ABB RAPID module: RapidProgrammeCode.mod

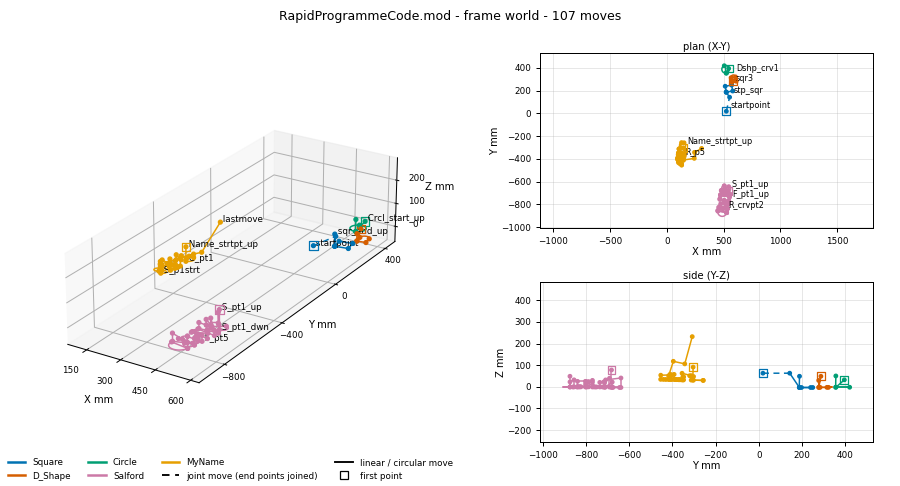
[picture p0: tool path of RapidProgrammeCode.mod in frame world, 107 of 113 moves have a stored position in this frame; points joined in program order, loops and branches not executed]
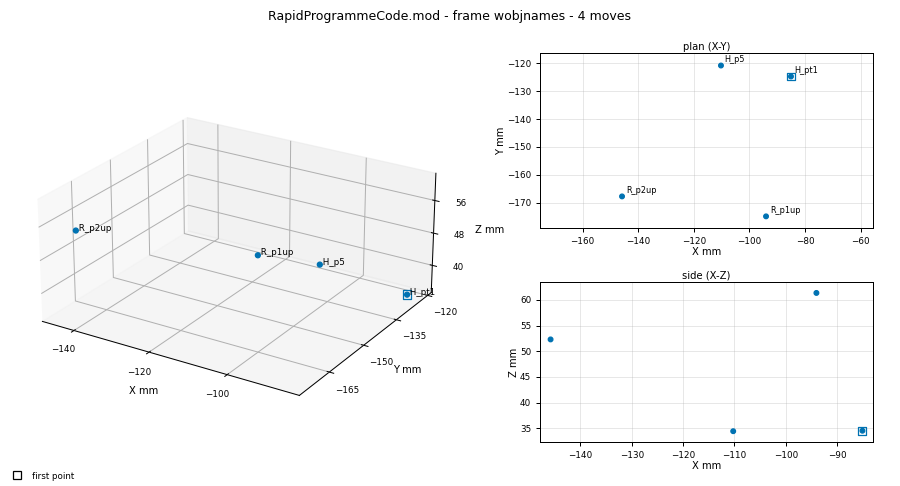
[picture p1: tool path of RapidProgrammeCode.mod in frame wobjnames, 4 of 113 moves have a stored position in this frame; points joined in program order, loops and branches not executed]
MODULE Module1
TASK PERS tooldata toolpen:=[TRUE,[[100,0,20],[1,0,0,0]],[0.1,[50,0,10],[1,0,0,0],0,0,0]];
TASK PERS wobjdata wobjshapes:=[FALSE,TRUE,"",[[456.883,136.274,-5.92371],[0.996185,0.000008375,-0.000001296,0.0872714]],[[0,0,0],[1,0,0,0]]];
CONST robtarget pointoforigin:=[[581.51,18.36,14.08],[0.66738,-0.167376,0.708898,0.155091],[-1,-1,0,1],[9E+9,9E+9,9E+9,9E+9,9E+9,9E+9]];
TASK PERS wobjdata wobjsalf:=[FALSE,TRUE,"",[[460.965,-385.411,-5.78367],[1,-0.000000822,-0.000000764,-0.000000546]],[[0,0,0],[1,0,0,0]]];
TASK PERS wobjdata wobjname:=[FALSE,TRUE,"",[[241.141,-193.884,-5.92118],[0.999813,-0.0119256,-0.000182929,0.0152539]],[[0,0,0],[1,0,0,0]]];
CONST robtarget startpoint:=[[45.66,-127.08,69.03],[0.678366,-0.104877,0.720803,0.0962504],[-1,-1,0,1],[9E+09,9E+09,9E+09,9E+09,9E+09,9E+09]];
CONST robtarget startpoint10:=[[105.53,42.34,81.65],[0.678367,-0.104876,0.720802,0.0962504],[0,-1,0,1],[9E+9,9E+9,9E+9,9E+9,9E+9,9E+9]];
CONST robtarget stp_sqr:=[[95.33,-10.14,69.03],[0.678365,-0.104877,0.720803,0.0962505],[0,-1,0,1],[9E+09,9E+09,9E+09,9E+09,9E+09,9E+09]];
CONST robtarget stp_sqr10:=[[72.90,39.01,0.49],[0.678366,-0.104876,0.720802,0.0962504],[0,-1,-1,1],[9E+9,9E+9,9E+9,9E+9,9E+9,9E+9]];
CONST robtarget stp_sqr1:=[[72.90,39.01,0.49],[0.678366,-0.104876,0.720802,0.0962504],[0,-1,-1,1],[9E+9,9E+9,9E+9,9E+9,9E+9,9E+9]];
CONST robtarget stp_sqr11:=[[131.10,38.55,0.49],[0.678367,-0.104876,0.720802,0.0962505],[0,-1,0,1],[9E+9,9E+9,9E+9,9E+9,9E+9,9E+9]];
CONST robtarget stp_sqr2:=[[131.10,38.55,0.49],[0.678367,-0.104876,0.720802,0.0962505],[0,-1,0,1],[9E+9,9E+9,9E+9,9E+9,9E+9,9E+9]];
CONST robtarget stp_sqr12:=[[130.95,91.71,0.49],[0.678366,-0.104876,0.720802,0.0962506],[0,-1,0,1],[9E+9,9E+9,9E+9,9E+9,9E+9,9E+9]];
CONST robtarget stp_sqr3:=[[130.95,91.71,0.49],[0.678366,-0.104876,0.720802,0.0962506],[0,-1,0,1],[9E+9,9E+9,9E+9,9E+9,9E+9,9E+9]];
CONST robtarget stp_sqr13:=[[72.83,91.46,0.49],[0.678365,-0.104877,0.720803,0.0962506],[0,-1,-1,1],[9E+9,9E+9,9E+9,9E+9,9E+9,9E+9]];
CONST robtarget stp_sqr4:=[[72.83,91.46,0.49],[0.678365,-0.104877,0.720803,0.0962506],[0,-1,-1,1],[9E+9,9E+9,9E+9,9E+9,9E+9,9E+9]];
CONST robtarget sqr1:=[[73.63,39.09,2.89],[0.678366,-0.104876,0.720803,0.0962505],[0,-1,-1,1],[9E+09,9E+09,9E+09,9E+09,9E+09,9E+09]];
CONST robtarget sqr2:=[[131.71,38.69,2.89],[0.678366,-0.104876,0.720803,0.0962504],[0,-1,0,1],[9E+09,9E+09,9E+09,9E+09,9E+09,9E+09]];
CONST robtarget sqr3:=[[131.6,91.52,2.89],[0.678365,-0.104877,0.720803,0.0962505],[0,-1,0,1],[9E+09,9E+09,9E+09,9E+09,9E+09,9E+09]];
CONST robtarget sqr4:=[[74.02,91.72,2.89],[0.678364,-0.104877,0.720805,0.0962503],[0,-1,-1,1],[9E+09,9E+09,9E+09,9E+09,9E+09,9E+09]];
CONST robtarget sqr14:=[[75.15,37.61,0.49],[0.678366,-0.104877,0.720803,0.0962507],[0,-1,-1,1],[9E+9,9E+9,9E+9,9E+9,9E+9,9E+9]];
CONST robtarget sqr24:=[[75.29,39.68,0.49],[0.678366,-0.104877,0.720803,0.0962508],[0,-1,-1,1],[9E+9,9E+9,9E+9,9E+9,9E+9,9E+9]];
CONST robtarget sqr5:=[[75.37,38.14,2.89],[0.678365,-0.104877,0.720804,0.0962503],[0,-1,-1,1],[9E+09,9E+09,9E+09,9E+09,9E+09,9E+09]];
CONST robtarget sqr15:=[[73.98,39.56,54.84],[0.678365,-0.104877,0.720803,0.0962503],[0,-1,0,1],[9E+9,9E+9,9E+9,9E+9,9E+9,9E+9]];
CONST robtarget sqr25:=[[73.98,39.56,54.84],[0.678365,-0.104877,0.720803,0.0962503],[0,-1,0,1],[9E+9,9E+9,9E+9,9E+9,9E+9,9E+9]];
CONST robtarget sqr_end_up:=[[73.98,39.56,54.84],[0.678365,-0.104877,0.720803,0.0962503],[0,-1,0,1],[9E+09,9E+09,9E+09,9E+09,9E+09,9E+09]];
CONST robtarget sqr_end_up10:=[[152.51,126.22,54.84],[0.678365,-0.104877,0.720804,0.0962505],[0,-1,-1,1],[9E+9,9E+9,9E+9,9E+9,9E+9,9E+9]];
CONST robtarget Dshp_start_up:=[[152.51,126.22,54.84],[0.678365,-0.104877,0.720804,0.0962505],[0,-1,-1,1],[9E+09,9E+09,9E+09,9E+09,9E+09,9E+09]];
CONST robtarget Dshp_start_up10:=[[139.65,118.70,3.57],[0.678364,-0.104877,0.720804,0.0962503],[0,-1,-1,1],[9E+9,9E+9,9E+9,9E+9,9E+9,9E+9]];
CONST robtarget Dshp_pt1:=[[139.65,118.7,3.57],[0.678364,-0.104877,0.720804,0.0962503],[0,-1,-1,1],[9E+09,9E+09,9E+09,9E+09,9E+09,9E+09]];
CONST robtarget Dshp_pt11:=[[177.47,117.91,3.57],[0.678365,-0.104877,0.720804,0.0962505],[0,-1,0,1],[9E+9,9E+9,9E+9,9E+9,9E+9,9E+9]];
CONST robtarget Dshp_pt2:=[[177.47,117.91,3.57],[0.678365,-0.104877,0.720804,0.0962505],[0,-1,0,1],[9E+09,9E+09,9E+09,9E+09,9E+09,9E+09]];
CONST robtarget Dshp_pt12:=[[177.53,157.32,3.57],[0.678364,-0.104877,0.720805,0.0962505],[0,0,-1,1],[9E+9,9E+9,9E+9,9E+9,9E+9,9E+9]];
CONST robtarget Dshp_pt3:=[[177.53,157.32,3.57],[0.678364,-0.104877,0.720805,0.0962505],[0,0,-1,1],[9E+09,9E+09,9E+09,9E+09,9E+09,9E+09]];
CONST robtarget Dshp_pt23:=[[138.50,156.89,3.57],[0.678363,-0.104877,0.720805,0.0962503],[0,0,-1,1],[9E+9,9E+9,9E+9,9E+9,9E+9,9E+9]];
CONST robtarget Dshp_pt13:=[[156.88,176.76,3.57],[0.678363,-0.104877,0.720805,0.0962503],[0,0,-1,1],[9E+9,9E+9,9E+9,9E+9,9E+9,9E+9]];
CONST robtarget Dshp_crv1:=[[156.88,176.76,3.57],[0.678363,-0.104877,0.720805,0.0962503],[0,0,-1,1],[9E+09,9E+09,9E+09,9E+09,9E+09,9E+09]];
CONST robtarget Dshp_crv2:=[[138.5,156.89,3.57],[0.678363,-0.104877,0.720805,0.0962503],[0,0,-1,1],[9E+09,9E+09,9E+09,9E+09,9E+09,9E+09]];
CONST robtarget Dshp_crv11:=[[139.05,118.30,3.57],[0.678363,-0.104877,0.720805,0.0962504],[0,-1,-1,1],[9E+9,9E+9,9E+9,9E+9,9E+9,9E+9]];
CONST robtarget Dshp_pt4:=[[139.05,118.3,3.57],[0.678363,-0.104877,0.720805,0.0962504],[0,-1,-1,1],[9E+09,9E+09,9E+09,9E+09,9E+09,9E+09]];
CONST robtarget Dshp_pt14:=[[139.05,118.30,35.44],[0.678363,-0.104877,0.720805,0.0962504],[0,-1,-1,1],[9E+9,9E+9,9E+9,9E+9,9E+9,9E+9]];
CONST robtarget Dshp_end_up:=[[139.05,118.3,35.44],[0.678363,-0.104877,0.720805,0.0962504],[0,-1,-1,1],[9E+09,9E+09,9E+09,9E+09,9E+09,9E+09]];
CONST robtarget Dshp_end_up10:=[[131.01,240.02,38.32],[0.678365,-0.104877,0.720803,0.0962513],[0,0,-1,1],[9E+9,9E+9,9E+9,9E+9,9E+9,9E+9]];
CONST robtarget Crcl_start_up:=[[131.01,240.02,38.32],[0.678365,-0.104877,0.720803,0.0962513],[0,0,-1,1],[9E+09,9E+09,9E+09,9E+09,9E+09,9E+09]];
CONST robtarget Crcl_start_up10:=[[104.28,205.24,4.07],[0.678363,-0.104878,0.720805,0.096251],[0,0,-1,1],[9E+9,9E+9,9E+9,9E+9,9E+9,9E+9]];
CONST robtarget Crcl_start_pt1:=[[104.28,205.24,4.07],[0.678363,-0.104878,0.720805,0.096251],[0,0,-1,1],[9E+09,9E+09,9E+09,9E+09,9E+09,9E+09]];
CONST robtarget Crcl_start_pt21:=[[97.32,270.88,4.07],[0.678363,-0.104878,0.720805,0.096251],[0,0,-1,1],[9E+9,9E+9,9E+9,9E+9,9E+9,9E+9]];
CONST robtarget Crcl_start_pt11:=[[134.47,246.88,4.07],[0.678363,-0.104878,0.720805,0.0962509],[0,0,-1,1],[9E+9,9E+9,9E+9,9E+9,9E+9,9E+9]];
CONST robtarget Crcl_pt2:=[[134.47,246.88,4.07],[0.678363,-0.104878,0.720805,0.0962509],[0,0,-1,1],[9E+09,9E+09,9E+09,9E+09,9E+09,9E+09]];
CONST robtarget Crcl_pt3:=[[97.32,270.88,4.07],[0.678363,-0.104878,0.720805,0.096251],[0,0,-1,1],[9E+09,9E+09,9E+09,9E+09,9E+09,9E+09]];
CONST robtarget Crcl_pt22:=[[104.26,203.85,4.07],[0.678363,-0.104878,0.720805,0.0962515],[0,0,-1,1],[9E+9,9E+9,9E+9,9E+9,9E+9,9E+9]];
CONST robtarget Crcl_pt12:=[[71.11,230.12,4.07],[0.678363,-0.104878,0.720805,0.0962513],[0,0,-1,1],[9E+9,9E+9,9E+9,9E+9,9E+9,9E+9]];
CONST robtarget Crcl_pt4:=[[71.11,230.12,4.07],[0.678363,-0.104878,0.720805,0.0962513],[0,0,-1,1],[9E+09,9E+09,9E+09,9E+09,9E+09,9E+09]];
CONST robtarget Crcl_pt5:=[[104.26,203.85,4.07],[0.678363,-0.104878,0.720805,0.0962515],[0,0,-1,1],[9E+09,9E+09,9E+09,9E+09,9E+09,9E+09]];
CONST robtarget Crcl_pt14:=[[103.87,204.92,56.32],[0.678365,-0.104876,0.720803,0.0962504],[0,0,-1,1],[9E+9,9E+9,9E+9,9E+9,9E+9,9E+9]];
CONST robtarget Crcl_end_up:=[[103.87,204.92,56.32],[0.678365,-0.104876,0.720803,0.0962504],[0,0,-1,1],[9E+09,9E+09,9E+09,9E+09,9E+09,9E+09]];
VAR num MyChoice:=0;
CONST robtarget Crcl_end_up10:=[[77.92,-295.75,83.77],[0.678363,-0.104878,0.720805,0.0962498],[-1,-1,0,1],[9E+9,9E+9,9E+9,9E+9,9E+9,9E+9]];
CONST robtarget S_pt1_up:=[[77.92,-295.75,83.77],[0.678363,-0.104878,0.720805,0.0962498],[-1,-1,0,1],[9E+09,9E+09,9E+09,9E+09,9E+09,9E+09]];
CONST robtarget S_pt1_up10:=[[77.92,-295.75,5.22],[0.678363,-0.104878,0.720805,0.0962496],[-1,-1,0,1],[9E+9,9E+9,9E+9,9E+9,9E+9,9E+9]];
CONST robtarget S_pt1_dwn:=[[77.92,-295.75,2.89],[0.678363,-0.104878,0.720805,0.0962498],[-1,-1,0,1],[9E+09,9E+09,9E+09,9E+09,9E+09,9E+09]];
CONST robtarget S_pt1_dwn20:=[[84.34,-258.56,5.22],[0.678363,-0.104877,0.720806,0.0962498],[-1,-1,0,1],[9E+9,9E+9,9E+9,9E+9,9E+9,9E+9]];
CONST robtarget S_pt1_dwn10:=[[100.17,-280.53,5.22],[0.678363,-0.104878,0.720805,0.0962498],[-1,-1,0,1],[9E+9,9E+9,9E+9,9E+9,9E+9,9E+9]];
CONST robtarget S_pt2_crv:=[[100.97,-278.71,2.9],[0.678364,-0.104879,0.720804,0.0962497],[-1,-1,0,1],[9E+09,9E+09,9E+09,9E+09,9E+09,9E+09]];
CONST robtarget S_pt2_crv2:=[[84.34,-258.56,5.22],[0.678363,-0.104877,0.720806,0.0962498],[-1,-1,0,1],[9E+9,9E+9,9E+9,9E+9,9E+9,9E+9]];
CONST robtarget S_pt2_crv10:=[[38.36,-288.97,5.22],[0.678362,-0.104877,0.720806,0.0962497],[-1,-1,0,1],[9E+9,9E+9,9E+9,9E+9,9E+9,9E+9]];
CONST robtarget S_pt3_crv2:=[[84.01,-258.59,2.9],[0.678364,-0.104878,0.720804,0.0962498],[-1,-1,0,1],[9E+09,9E+09,9E+09,9E+09,9E+09,9E+09]];
CONST robtarget S_pt4:=[[40.74,-288.86,2.9],[0.678364,-0.104878,0.720804,0.0962498],[-1,-1,0,1],[9E+09,9E+09,9E+09,9E+09,9E+09,9E+09]];
CONST robtarget S_pt24:=[[44.83,-251.34,5.22],[0.678362,-0.104877,0.720806,0.0962497],[-1,-1,0,1],[9E+9,9E+9,9E+9,9E+9,9E+9,9E+9]];
CONST robtarget S_pt14:=[[22.78,-267.45,5.22],[0.678362,-0.104877,0.720806,0.0962498],[-1,-1,0,1],[9E+9,9E+9,9E+9,9E+9,9E+9,9E+9]];
CONST robtarget S_pt5_crv3:=[[22.75,-267.87,2.89],[0.678363,-0.104878,0.720805,0.0962498],[-1,-1,0,1],[9E+09,9E+09,9E+09,9E+09,9E+09,9E+09]];
CONST robtarget S_pt6_crv4:=[[44.86,-252.05,2.89],[0.678363,-0.104878,0.720805,0.09625],[-1,-1,0,1],[9E+09,9E+09,9E+09,9E+09,9E+09,9E+09]];
CONST robtarget S_pt5_crv13:=[[44.83,-251.34,37.85],[0.678362,-0.104877,0.720806,0.0962496],[-1,-1,0,1],[9E+9,9E+9,9E+9,9E+9,9E+9,9E+9]];
CONST robtarget S_end_up:=[[44.86,-252.05,46.77],[0.678363,-0.104878,0.720805,0.09625],[-1,-1,0,1],[9E+09,9E+09,9E+09,9E+09,9E+09,9E+09]];
CONST robtarget S_end_up10:=[[92.49,-322.94,37.85],[0.678363,-0.104877,0.720806,0.0962493],[-1,-1,0,1],[9E+9,9E+9,9E+9,9E+9,9E+9,9E+9]];
CONST robtarget S_end_up20:=[[92.49,-322.94,37.85],[0.678363,-0.104877,0.720806,0.0962493],[-1,-1,0,1],[9E+9,9E+9,9E+9,9E+9,9E+9,9E+9]];
CONST robtarget A_start_up:=[[92.49,-322.94,37.85],[0.678363,-0.104877,0.720806,0.0962493],[-1,-1,0,1],[9E+09,9E+09,9E+09,9E+09,9E+09,9E+09]];
CONST robtarget A_start_up10:=[[91.38,-324.75,5.35],[0.678363,-0.104877,0.720806,0.0962492],[-1,-1,0,1],[9E+9,9E+9,9E+9,9E+9,9E+9,9E+9]];
CONST robtarget A_start_pt1:=[[91.38,-324.75,5.35],[0.678363,-0.104877,0.720806,0.0962492],[-1,-1,0,1],[9E+09,9E+09,9E+09,9E+09,9E+09,9E+09]];
CONST robtarget A_start_pt11:=[[18.61,-292.43,5.35],[0.678364,-0.104878,0.720805,0.0962491],[-1,-1,0,1],[9E+9,9E+9,9E+9,9E+9,9E+9,9E+9]];
CONST robtarget A_pt2:=[[18.61,-292.43,5.35],[0.678364,-0.104878,0.720805,0.0962491],[-1,-1,0,1],[9E+09,9E+09,9E+09,9E+09,9E+09,9E+09]];
CONST robtarget A_pt12:=[[18.61,-292.43,27.82],[0.678364,-0.104877,0.720805,0.096249],[-1,-1,0,1],[9E+9,9E+9,9E+9,9E+9,9E+9,9E+9]];
CONST robtarget A_line1_up:=[[18.61,-292.43,27.82],[0.678364,-0.104877,0.720805,0.096249],[-1,-1,0,1],[9E+09,9E+09,9E+09,9E+09,9E+09,9E+09]];
CONST robtarget A_line1_up10:=[[91.72,-324.34,4.75],[0.678363,-0.104878,0.720806,0.0962488],[-1,-1,0,1],[9E+9,9E+9,9E+9,9E+9,9E+9,9E+9]];
CONST robtarget A_line2_strt:=[[91.72,-324.34,4.75],[0.678363,-0.104878,0.720806,0.0962488],[-1,-1,0,1],[9E+09,9E+09,9E+09,9E+09,9E+09,9E+09]];
CONST robtarget A_line2_strt10:=[[11.68,-330.33,4.75],[0.678362,-0.104877,0.720806,0.096249],[-1,-1,0,1],[9E+9,9E+9,9E+9,9E+9,9E+9,9E+9]];
CONST robtarget A_line2_stp:=[[11.68,-330.33,4.75],[0.678362,-0.104877,0.720806,0.096249],[-1,-1,0,1],[9E+09,9E+09,9E+09,9E+09,9E+09,9E+09]];
CONST robtarget A_line2_stp10:=[[11.68,-330.33,29.04],[0.678362,-0.104877,0.720806,0.0962488],[-1,-1,0,1],[9E+9,9E+9,9E+9,9E+9,9E+9,9E+9]];
CONST robtarget A_line2_endup:=[[11.68,-330.33,29.04],[0.678362,-0.104877,0.720806,0.0962488],[-1,-1,0,1],[9E+09,9E+09,9E+09,9E+09,9E+09,9E+09]];
CONST robtarget A_line2_endup10:=[[43.93,-327.74,25.23],[0.678361,-0.104877,0.720807,0.0962489],[-1,-1,0,1],[9E+9,9E+9,9E+9,9E+9,9E+9,9E+9]];
CONST robtarget A_crssline_up:=[[43.93,-327.74,25.23],[0.678361,-0.104877,0.720807,0.0962489],[-1,-1,0,1],[9E+09,9E+09,9E+09,9E+09,9E+09,9E+09]];
CONST robtarget A_crssline_up10:=[[43.93,-327.74,4.82],[0.678361,-0.104878,0.720807,0.0962489],[-1,-1,0,1],[9E+9,9E+9,9E+9,9E+9,9E+9,9E+9]];
CONST robtarget A_crssline_pt1:=[[43.93,-327.74,4.82],[0.678361,-0.104878,0.720807,0.0962489],[-1,-1,0,1],[9E+09,9E+09,9E+09,9E+09,9E+09,9E+09]];
CONST robtarget A_crssline_pt11:=[[46.49,-305.03,4.82],[0.678361,-0.104878,0.720808,0.0962489],[-1,-1,0,1],[9E+9,9E+9,9E+9,9E+9,9E+9,9E+9]];
CONST robtarget A_crssline_pt2:=[[46.49,-305.03,4.82],[0.67836,-0.104878,0.720808,0.096249],[-1,-1,0,1],[9E+09,9E+09,9E+09,9E+09,9E+09,9E+09]];
CONST robtarget A_crssline_pt12:=[[46.49,-305.03,45.39],[0.67836,-0.104878,0.720808,0.0962488],[-1,-1,0,1],[9E+9,9E+9,9E+9,9E+9,9E+9,9E+9]];
CONST robtarget A_end_up:=[[46.49,-305.03,45.39],[0.67836,-0.104878,0.720808,0.0962488],[-1,-1,0,1],[9E+09,9E+09,9E+09,9E+09,9E+09,9E+09]];
CONST robtarget A_end_up10:=[[91.77,-349.30,45.39],[0.678361,-0.104878,0.720808,0.0962487],[-1,-1,0,1],[9E+9,9E+9,9E+9,9E+9,9E+9,9E+9]];
CONST robtarget L_start_up:=[[90.88,-349.88,26.27],[0.67836,-0.104879,0.720808,0.0962479],[-1,-1,0,1],[9E+09,9E+09,9E+09,9E+09,9E+09,9E+09]];
CONST robtarget L_start_up10:=[[89.10,-349.57,5.90],[0.67836,-0.104878,0.720808,0.0962488],[-1,-1,0,1],[9E+9,9E+9,9E+9,9E+9,9E+9,9E+9]];
CONST robtarget L_start_pt1:=[[90.88,-349.88,5.25],[0.67836,-0.104879,0.720809,0.0962479],[-1,-1,0,1],[9E+09,9E+09,9E+09,9E+09,9E+09,9E+09]];
CONST robtarget L_start_pt11:=[[11.36,-337.10,5.90],[0.67836,-0.104878,0.720808,0.0962488],[-1,-1,0,1],[9E+9,9E+9,9E+9,9E+9,9E+9,9E+9]];
CONST robtarget L_pt2:=[[11.36,-337.10,5.90],[0.67836,-0.104878,0.720808,0.0962488],[-1,-1,0,1],[9E+9,9E+9,9E+9,9E+9,9E+9,9E+9]];
CONST robtarget L_pt3_dwn:=[[11.26,-336.76,5.25],[0.67836,-0.104879,0.720809,0.0962477],[-1,-1,0,1],[9E+09,9E+09,9E+09,9E+09,9E+09,9E+09]];
CONST robtarget L_pt3_dwn10:=[[6.45,-364.89,29.17],[0.678361,-0.104878,0.720808,0.0962485],[-1,-1,0,1],[9E+9,9E+9,9E+9,9E+9,9E+9,9E+9]];
CONST robtarget L_pt3_up:=[[6.26,-365.07,5.25],[0.67836,-0.104879,0.720808,0.0962476],[-1,-1,0,1],[9E+9,9E+9,9E+9,9E+9,9E+9,9E+9]];
CONST robtarget L_pt3_up10:=[[82.67,-383.82,35.68],[0.678359,-0.104878,0.720809,0.0962486],[-1,-1,0,1],[9E+9,9E+9,9E+9,9E+9,9E+9,9E+9]];
CONST robtarget F_pt1_up:=[[82.67,-383.82,35.68],[0.678359,-0.104878,0.720809,0.0962486],[-1,-1,0,1],[9E+09,9E+09,9E+09,9E+09,9E+09,9E+09]];
CONST robtarget F_pt1_up10:=[[82.67,-383.82,5.13],[0.678359,-0.104879,0.720809,0.0962485],[-1,-1,0,1],[9E+9,9E+9,9E+9,9E+9,9E+9,9E+9]];
CONST robtarget F_pt1_dwn:=[[82.67,-383.82,5.13],[0.678359,-0.104879,0.720809,0.0962485],[-1,-1,0,1],[9E+09,9E+09,9E+09,9E+09,9E+09,9E+09]];
CONST robtarget F_pt1_dwn10:=[[5.32,-370.91,5.13],[0.678359,-0.104878,0.720809,0.0962484],[-1,-1,0,1],[9E+9,9E+9,9E+9,9E+9,9E+9,9E+9]];
CONST robtarget F_pt2:=[[5.32,-370.91,5.13],[0.678359,-0.104878,0.720809,0.0962484],[-1,-1,0,1],[9E+09,9E+09,9E+09,9E+09,9E+09,9E+09]];
CONST robtarget F_pt12:=[[84.74,-384.03,26.67],[0.678359,-0.104878,0.720809,0.0962485],[-1,-1,0,1],[9E+9,9E+9,9E+9,9E+9,9E+9,9E+9]];
CONST robtarget F_pt3:=[[84.74,-384.03,26.67],[0.678359,-0.104878,0.720809,0.0962485],[-1,-1,0,1],[9E+09,9E+09,9E+09,9E+09,9E+09,9E+09]];
CONST robtarget F_pt13:=[[83.30,-383.78,5.09],[0.678358,-0.104878,0.72081,0.0962484],[-1,-1,0,1],[9E+9,9E+9,9E+9,9E+9,9E+9,9E+9]];
CONST robtarget F_pt4:=[[83.3,-383.78,5.09],[0.678358,-0.104878,0.72081,0.0962484],[-1,-1,0,1],[9E+09,9E+09,9E+09,9E+09,9E+09,9E+09]];
CONST robtarget F_pt14:=[[78.23,-412.54,5.09],[0.678359,-0.104878,0.720809,0.0962483],[-1,-1,0,1],[9E+9,9E+9,9E+9,9E+9,9E+9,9E+9]];
CONST robtarget F_pt5:=[[78.23,-412.54,5.09],[0.678359,-0.104878,0.720809,0.0962483],[-1,-1,0,1],[9E+09,9E+09,9E+09,9E+09,9E+09,9E+09]];
CONST robtarget F_pt15:=[[78.23,-412.54,29.87],[0.678359,-0.104878,0.72081,0.0962482],[-1,-1,0,1],[9E+9,9E+9,9E+9,9E+9,9E+9,9E+9]];
CONST robtarget F_pt5_up:=[[78.23,-412.54,29.87],[0.678359,-0.104878,0.72081,0.0962482],[-1,-1,0,1],[9E+09,9E+09,9E+09,9E+09,9E+09,9E+09]];
CONST robtarget F_pt5_up10:=[[44.03,-377.25,5.78],[0.678357,-0.104877,0.720811,0.0962484],[-1,-1,0,1],[9E+9,9E+9,9E+9,9E+9,9E+9,9E+9]];
CONST robtarget F_pt6:=[[44.03,-377.25,5.78],[0.678357,-0.104877,0.720811,0.0962484],[-1,-1,0,1],[9E+09,9E+09,9E+09,9E+09,9E+09,9E+09]];
CONST robtarget F_pt16:=[[40.82,-401.74,5.78],[0.678358,-0.104878,0.72081,0.0962483],[-1,-1,0,1],[9E+9,9E+9,9E+9,9E+9,9E+9,9E+9]];
CONST robtarget F_pt7_enddwn:=[[40.82,-401.74,5.78],[0.678358,-0.104878,0.72081,0.0962483],[-1,-1,0,1],[9E+09,9E+09,9E+09,9E+09,9E+09,9E+09]];
CONST robtarget F_pt7_enddwn10:=[[40.82,-401.74,30.12],[0.678358,-0.104877,0.72081,0.096248],[-1,-1,0,1],[9E+9,9E+9,9E+9,9E+9,9E+9,9E+9]];
CONST robtarget F_pt7_endup:=[[40.82,-401.74,30.12],[0.678358,-0.104877,0.72081,0.096248],[-1,-1,0,1],[9E+09,9E+09,9E+09,9E+09,9E+09,9E+09]];
CONST robtarget F_pt7_endup10:=[[62.72,-415.58,18.75],[0.678357,-0.104876,0.720811,0.0962485],[-1,-1,0,1],[9E+9,9E+9,9E+9,9E+9,9E+9,9E+9]];
CONST robtarget O_pt1_strtup:=[[62.72,-415.58,18.75],[0.678357,-0.104876,0.720811,0.0962485],[-1,-1,0,1],[9E+09,9E+09,9E+09,9E+09,9E+09,9E+09]];
CONST robtarget O_pt1_strtup10:=[[62.63,-416.14,5.89],[0.678357,-0.104877,0.720811,0.0962485],[-1,-1,0,1],[9E+9,9E+9,9E+9,9E+9,9E+9,9E+9]];
CONST robtarget O_pt1_dwn:=[[62.63,-416.14,5.89],[0.678357,-0.104877,0.720811,0.0962485],[-1,-1,0,1],[9E+09,9E+09,9E+09,9E+09,9E+09,9E+09]];
CONST robtarget O_pt1_dwn20:=[[59.21,-444.89,5.90],[0.678358,-0.104878,0.72081,0.0962479],[-1,-1,0,1],[9E+9,9E+9,9E+9,9E+9,9E+9,9E+9]];
CONST robtarget O_pt1_dwn10:=[[75.48,-430.52,5.90],[0.678358,-0.104878,0.72081,0.0962483],[-1,-1,0,1],[9E+9,9E+9,9E+9,9E+9,9E+9,9E+9]];
CONST robtarget O_crv1:=[[75.48,-430.52,5.9],[0.678358,-0.104878,0.72081,0.0962483],[-1,-1,0,1],[9E+09,9E+09,9E+09,9E+09,9E+09,9E+09]];
CONST robtarget O_crv2:=[[59.21,-444.89,5.9],[0.678358,-0.104878,0.72081,0.0962479],[-1,-1,0,1],[9E+09,9E+09,9E+09,9E+09,9E+09,9E+09]];
CONST robtarget O_crv11:=[[10.66,-437.03,5.90],[0.678359,-0.104877,0.72081,0.0962477],[-1,-1,0,1],[9E+9,9E+9,9E+9,9E+9,9E+9,9E+9]];
CONST robtarget O_pt2:=[[10.66,-437.03,5.9],[0.678359,-0.104877,0.72081,0.0962477],[-1,-1,0,1],[9E+09,9E+09,9E+09,9E+09,9E+09,9E+09]];
CONST robtarget O_pt22:=[[13.68,-408.53,5.90],[0.678358,-0.104877,0.72081,0.0962479],[-1,-1,0,1],[9E+9,9E+9,9E+9,9E+9,9E+9,9E+9]];
CONST robtarget O_pt12:=[[-1.80,-420.36,5.90],[0.678358,-0.104877,0.720811,0.0962481],[-1,-1,0,1],[9E+9,9E+9,9E+9,9E+9,9E+9,9E+9]];
CONST robtarget O_crv3:=[[-1.8,-420.36,5.9],[0.678358,-0.104877,0.720811,0.0962481],[-1,-1,0,1],[9E+09,9E+09,9E+09,9E+09,9E+09,9E+09]];
CONST robtarget O_crv4:=[[13.68,-408.53,5.9],[0.678358,-0.104877,0.72081,0.0962479],[-1,-1,0,1],[9E+09,9E+09,9E+09,9E+09,9E+09,9E+09]];
CONST robtarget O_crv13:=[[62.31,-416.42,5.90],[0.678358,-0.104878,0.72081,0.0962481],[-1,-1,0,1],[9E+9,9E+9,9E+9,9E+9,9E+9,9E+9]];
CONST robtarget O_endpt_dwn:=[[62.31,-416.42,5.9],[0.678358,-0.104878,0.72081,0.0962481],[-1,-1,0,1],[9E+09,9E+09,9E+09,9E+09,9E+09,9E+09]];
CONST robtarget O_endpt_dwn10:=[[62.31,-416.42,31.24],[0.678358,-0.104877,0.72081,0.0962481],[-1,-1,0,1],[9E+9,9E+9,9E+9,9E+9,9E+9,9E+9]];
CONST robtarget O_endpt_up:=[[62.31,-416.42,31.24],[0.678358,-0.104877,0.72081,0.0962481],[-1,-1,0,1],[9E+09,9E+09,9E+09,9E+09,9E+09,9E+09]];
CONST robtarget O_endpt_up10:=[[72.94,-452.85,31.24],[0.678357,-0.104876,0.720811,0.096249],[-1,-1,0,1],[9E+9,9E+9,9E+9,9E+9,9E+9,9E+9]];
CONST robtarget R_strtpt_up:=[[72.94,-452.85,31.24],[0.678357,-0.104876,0.720811,0.096249],[-1,-1,0,1],[9E+09,9E+09,9E+09,9E+09,9E+09,9E+09]];
CONST robtarget R_strtpt_up10:=[[72.09,-452.79,6.00],[0.678357,-0.104877,0.720811,0.0962489],[-1,-1,0,1],[9E+9,9E+9,9E+9,9E+9,9E+9,9E+9]];
CONST robtarget R_strt_pt1:=[[72.09,-452.79,6],[0.678357,-0.104877,0.720811,0.0962489],[-1,-1,0,1],[9E+09,9E+09,9E+09,9E+09,9E+09,9E+09]];
CONST robtarget R_strt_pt11:=[[-4.81,-440.43,6.00],[0.678357,-0.104877,0.720811,0.0962487],[-1,-1,0,1],[9E+9,9E+9,9E+9,9E+9,9E+9,9E+9]];
CONST robtarget R_pt2:=[[-4.81,-440.43,6],[0.678357,-0.104877,0.720811,0.0962487],[-1,-1,0,1],[9E+09,9E+09,9E+09,9E+09,9E+09,9E+09]];
CONST robtarget R_pt12:=[[71.63,-452.78,5.74],[0.678356,-0.104876,0.720812,0.0962494],[-1,-1,0,1],[9E+9,9E+9,9E+9,9E+9,9E+9,9E+9]];
CONST robtarget R_crvpt1:=[[71.63,-452.78,5.74],[0.678356,-0.104876,0.720812,0.0962494],[-1,-1,0,1],[9E+09,9E+09,9E+09,9E+09,9E+09,9E+09]];
CONST robtarget R_crvpt21:=[[33.40,-446.98,5.74],[0.678356,-0.104875,0.720813,0.0962493],[-1,-1,0,1],[9E+9,9E+9,9E+9,9E+9,9E+9,9E+9]];
CONST robtarget R_crvpt11:=[[48.38,-478.62,5.74],[0.678356,-0.104876,0.720812,0.0962494],[-1,-1,0,1],[9E+9,9E+9,9E+9,9E+9,9E+9,9E+9]];
CONST robtarget R_crvpt2:=[[48.38,-478.62,5.74],[0.678356,-0.104876,0.720812,0.0962494],[-1,-1,0,1],[9E+09,9E+09,9E+09,9E+09,9E+09,9E+09]];
CONST robtarget R_crvpt3:=[[33.4,-446.98,5.74],[0.678356,-0.104875,0.720813,0.0962493],[-1,-1,0,1],[9E+09,9E+09,9E+09,9E+09,9E+09,9E+09]];
CONST robtarget R_crvpt12:=[[31.87,-455.63,5.45],[0.678356,-0.104875,0.720813,0.0962491],[-1,-1,0,1],[9E+9,9E+9,9E+9,9E+9,9E+9,9E+9]];
CONST robtarget R_endline1:=[[31.87,-455.63,5.45],[0.678356,-0.104875,0.720813,0.0962491],[-1,-1,0,1],[9E+09,9E+09,9E+09,9E+09,9E+09,9E+09]];
CONST robtarget R_endline11:=[[-11.14,-468.97,5.45],[0.678355,-0.104875,0.720813,0.0962493],[-1,-1,0,1],[9E+9,9E+9,9E+9,9E+9,9E+9,9E+9]];
CONST robtarget R_endline2:=[[-11.14,-468.97,5.45],[0.678355,-0.104875,0.720813,0.0962493],[-1,-1,0,1],[9E+09,9E+09,9E+09,9E+09,9E+09,9E+09]];
CONST robtarget R_endline12:=[[-11.14,-468.97,38.13],[0.678355,-0.104875,0.720813,0.0962491],[-1,-1,0,1],[9E+9,9E+9,9E+9,9E+9,9E+9,9E+9]];
CONST robtarget R_endline_up:=[[-11.14,-468.97,38.13],[0.678355,-0.104875,0.720813,0.0962491],[-1,-1,0,1],[9E+09,9E+09,9E+09,9E+09,9E+09,9E+09]];
CONST robtarget R_endline_up10:=[[66.05,-487.59,28.57],[0.678355,-0.104875,0.720813,0.0962494],[-1,-1,0,1],[9E+9,9E+9,9E+9,9E+9,9E+9,9E+9]];
CONST robtarget D_strt_up:=[[66.05,-487.59,28.57],[0.678355,-0.104875,0.720813,0.0962494],[-1,-1,0,1],[9E+09,9E+09,9E+09,9E+09,9E+09,9E+09]];
CONST robtarget D_strt_up10:=[[65.69,-487.52,5.12],[0.678354,-0.104875,0.720814,0.0962494],[-1,-1,0,1],[9E+9,9E+9,9E+9,9E+9,9E+9,9E+9]];
CONST robtarget D_pt1:=[[65.69,-487.52,5.12],[0.678354,-0.104875,0.720814,0.0962494],[-1,-1,0,1],[9E+09,9E+09,9E+09,9E+09,9E+09,9E+09]];
CONST robtarget D_pt11:=[[-11.81,-474.59,5.12],[0.678354,-0.104875,0.720814,0.0962493],[-1,-1,0,1],[9E+9,9E+9,9E+9,9E+9,9E+9,9E+9]];
CONST robtarget D_pt2:=[[-11.81,-474.59,5.12],[0.678354,-0.104875,0.720814,0.0962493],[-1,-1,0,1],[9E+09,9E+09,9E+09,9E+09,9E+09,9E+09]];
CONST robtarget D_pt22:=[[65.48,-487.84,5.12],[0.678354,-0.104875,0.720815,0.0962493],[-1,-1,0,1],[9E+9,9E+9,9E+9,9E+9,9E+9,9E+9]];
CONST robtarget D_pt12:=[[20.28,-519.61,5.12],[0.678354,-0.104875,0.720814,0.0962491],[-1,-1,0,1],[9E+9,9E+9,9E+9,9E+9,9E+9,9E+9]];
CONST robtarget D_crvpt1:=[[20.28,-519.61,5.12],[0.678354,-0.104875,0.720814,0.0962491],[-1,-1,0,1],[9E+09,9E+09,9E+09,9E+09,9E+09,9E+09]];
CONST robtarget D_crvpt2_end:=[[65.48,-487.84,5.12],[0.678354,-0.104875,0.720815,0.0962493],[-1,-1,0,1],[9E+09,9E+09,9E+09,9E+09,9E+09,9E+09]];
CONST robtarget D_crvpt11:=[[65.48,-487.84,54.70],[0.678354,-0.104875,0.720814,0.0962491],[-1,-1,0,1],[9E+9,9E+9,9E+9,9E+9,9E+9,9E+9]];
CONST robtarget D_end_up:=[[65.48,-487.84,54.7],[0.678354,-0.104875,0.720814,0.0962491],[-1,-1,0,1],[9E+09,9E+09,9E+09,9E+09,9E+09,9E+09]];
CONST robtarget L_end_pt4:=[[6.26,-365.07,5.25],[0.67836,-0.104879,0.720808,0.0962476],[-1,-1,0,1],[9E+09,9E+09,9E+09,9E+09,9E+09,9E+09]];
CONST robtarget L_end_pt14:=[[6.26,-365.07,37.03],[0.67836,-0.104879,0.720808,0.0962477],[-1,-1,0,1],[9E+9,9E+9,9E+9,9E+9,9E+9,9E+9]];
CONST robtarget L_end_ptup:=[[6.26,-365.07,37.03],[0.67836,-0.104879,0.720808,0.0962477],[-1,-1,0,1],[9E+09,9E+09,9E+09,9E+09,9E+09,9E+09]];
CONST robtarget D_end_up10:=[[-142.53,-93.79,88.23],[0.673249,0.302219,0.646493,-0.193511],[0,0,0,1],[9E+9,9E+9,9E+9,9E+9,9E+9,9E+9]];
CONST robtarget Name_strtpt_up:=[[-97.58,-109.23,94.65],[0.673249,0.302219,0.646493,-0.193511],[0,0,0,1],[9E+09,9E+09,9E+09,9E+09,9E+09,9E+09]];
CONST robtarget Name_strtpt_up10:=[[-142.53,-93.79,35.10],[0.673249,0.302219,0.646494,-0.193511],[0,0,0,1],[9E+9,9E+9,9E+9,9E+9,9E+9,9E+9]];
CONST robtarget C_pt1:=[[-97.58,-109.23,34.31],[0.673249,0.302219,0.646493,-0.193511],[0,0,0,1],[9E+09,9E+09,9E+09,9E+09,9E+09,9E+09]];
CONST robtarget C_pt21:=[[-143.69,-45.53,34.71],[0.673249,0.302219,0.646493,-0.19351],[0,0,0,1],[9E+9,9E+9,9E+9,9E+9,9E+9,9E+9]];
CONST robtarget C_pt11:=[[-123.31,-68.73,34.71],[0.673249,0.302218,0.646493,-0.19351],[0,0,0,1],[9E+9,9E+9,9E+9,9E+9,9E+9,9E+9]];
CONST robtarget C_pt2:=[[-77.64,-82.24,34.31],[0.673248,0.302219,0.646493,-0.193511],[0,0,0,1],[9E+09,9E+09,9E+09,9E+09,9E+09,9E+09]];
CONST robtarget C_pt3:=[[-91.37,-62.23,34.31],[0.673249,0.302218,0.646493,-0.193511],[0,0,0,1],[9E+09,9E+09,9E+09,9E+09,9E+09,9E+09]];
CONST robtarget C_pt22:=[[-175.30,-60.76,34.71],[0.673249,0.302219,0.646493,-0.19351],[0,0,0,1],[9E+9,9E+9,9E+9,9E+9,9E+9,9E+9]];
CONST robtarget C_pt12:=[[-175.30,-60.76,34.71],[0.673249,0.302219,0.646493,-0.19351],[0,0,0,1],[9E+9,9E+9,9E+9,9E+9,9E+9,9E+9]];
CONST robtarget C_pt4:=[[-175.30,-60.76,34.71],[0.673249,0.302219,0.646493,-0.19351],[0,0,0,1],[9E+9,9E+9,9E+9,9E+9,9E+9,9E+9]];
CONST robtarget C_pt5:=[[-165.50,-90.40,34.71],[0.673248,0.302218,0.646494,-0.19351],[0,0,0,1],[9E+9,9E+9,9E+9,9E+9,9E+9,9E+9]];
CONST robtarget C_pt14:=[[-165.50,-90.40,65.98],[0.673249,0.302218,0.646494,-0.19351],[0,0,0,1],[9E+9,9E+9,9E+9,9E+9,9E+9,9E+9]];
CONST robtarget C_endup:=[[-165.50,-90.40,65.98],[0.673249,0.302218,0.646494,-0.19351],[0,0,0,1],[9E+9,9E+9,9E+9,9E+9,9E+9,9E+9]];
CONST robtarget C_endup10:=[[-132.10,-114.55,65.98],[0.673249,0.302219,0.646494,-0.19351],[0,0,0,1],[9E+9,9E+9,9E+9,9E+9,9E+9,9E+9]];
CONST robtarget H_strtup:=[[-132.10,-114.55,65.98],[0.673249,0.302219,0.646494,-0.19351],[0,0,0,1],[9E+9,9E+9,9E+9,9E+9,9E+9,9E+9]];
CONST robtarget C_pt32:=[[-113.17,-60.06,34.31],[0.673249,0.30222,0.646493,-0.19351],[0,0,0,1],[9E+9,9E+9,9E+9,9E+9,9E+9,9E+9]];
CONST robtarget C_p4:=[[-113.17,-60.06,34.31],[0.673249,0.30222,0.646493,-0.19351],[0,0,0,1],[9E+09,9E+09,9E+09,9E+09,9E+09,9E+09]];
CONST robtarget C_p24:=[[-120.60,-105.61,34.31],[0.673249,0.30222,0.646492,-0.193511],[0,0,0,1],[9E+9,9E+9,9E+9,9E+9,9E+9,9E+9]];
CONST robtarget C_p14:=[[-131.25,-78.78,34.31],[0.673249,0.30222,0.646492,-0.19351],[0,0,0,1],[9E+9,9E+9,9E+9,9E+9,9E+9,9E+9]];
CONST robtarget C_p5:=[[-131.25,-78.78,34.31],[0.673249,0.30222,0.646492,-0.19351],[0,0,0,1],[9E+09,9E+09,9E+09,9E+09,9E+09,9E+09]];
CONST robtarget C_p6:=[[-120.6,-105.61,34.31],[0.673249,0.30222,0.646492,-0.193511],[0,0,0,1],[9E+09,9E+09,9E+09,9E+09,9E+09,9E+09]];
CONST robtarget C_p15:=[[-120.60,-105.61,51.11],[0.673249,0.30222,0.646493,-0.193511],[0,0,0,1],[9E+9,9E+9,9E+9,9E+9,9E+9,9E+9]];
CONST robtarget C_end_up:=[[-120.6,-105.61,51.11],[0.673249,0.30222,0.646493,-0.193511],[0,0,0,1],[9E+09,9E+09,9E+09,9E+09,9E+09,9E+09]];
CONST robtarget C_end_up10:=[[-85.09,-124.69,54.44],[0.673249,0.30222,0.646493,-0.193511],[0,0,0,1],[9E+9,9E+9,9E+9,9E+9,9E+9,9E+9]];
CONST robtarget H_startup:=[[-85.09,-124.69,54.44],[0.673249,0.30222,0.646493,-0.193511],[0,0,0,1],[9E+09,9E+09,9E+09,9E+09,9E+09,9E+09]];
CONST robtarget H_startup10:=[[-85.09,-124.69,34.51],[0.673248,0.30222,0.646493,-0.19351],[0,0,0,1],[9E+9,9E+9,9E+9,9E+9,9E+9,9E+9]];
CONST robtarget H_pt1:=[[-85.09,-124.69,34.51],[0.673248,0.30222,0.646493,-0.19351],[0,0,0,1],[9E+09,9E+09,9E+09,9E+09,9E+09,9E+09]];
CONST robtarget H_pt11:=[[-137.25,-115.48,34.51],[0.673248,0.30222,0.646493,-0.193511],[0,0,0,1],[9E+9,9E+9,9E+9,9E+9,9E+9,9E+9]];
CONST robtarget H_pt2:=[[-137.25,-115.48,34.51],[0.673248,0.30222,0.646493,-0.193511],[0,0,0,1],[9E+09,9E+09,9E+09,9E+09,9E+09,9E+09]];
CONST robtarget H_pt12:=[[-137.25,-115.48,54.91],[0.673248,0.30222,0.646493,-0.193511],[0,0,0,1],[9E+9,9E+9,9E+9,9E+9,9E+9,9E+9]];
CONST robtarget H_p2up:=[[-137.25,-115.48,54.91],[0.673248,0.30222,0.646493,-0.193511],[0,0,0,1],[9E+09,9E+09,9E+09,9E+09,9E+09,9E+09]];
CONST robtarget H_p2up10:=[[-91.33,-159.94,64.95],[0.673248,0.30222,0.646494,-0.193511],[0,0,0,1],[9E+9,9E+9,9E+9,9E+9,9E+9,9E+9]];
CONST robtarget H_p3up:=[[-91.33,-159.94,64.95],[0.673248,0.30222,0.646494,-0.193511],[0,0,0,1],[9E+09,9E+09,9E+09,9E+09,9E+09,9E+09]];
CONST robtarget H_p3up10:=[[-91.33,-159.94,34.41],[0.673248,0.30222,0.646494,-0.193511],[0,0,0,1],[9E+9,9E+9,9E+9,9E+9,9E+9,9E+9]];
CONST robtarget H_p3:=[[-91.33,-159.94,34.41],[0.673248,0.30222,0.646494,-0.193511],[0,0,0,1],[9E+09,9E+09,9E+09,9E+09,9E+09,9E+09]];
CONST robtarget H_p13:=[[-143.89,-150.66,34.41],[0.673248,0.30222,0.646494,-0.193511],[0,0,0,1],[9E+9,9E+9,9E+9,9E+9,9E+9,9E+9]];
CONST robtarget H_p4:=[[-143.89,-150.66,34.41],[0.673248,0.30222,0.646494,-0.193511],[0,0,0,1],[9E+09,9E+09,9E+09,9E+09,9E+09,9E+09]];
CONST robtarget H_p14:=[[-143.89,-150.66,48.70],[0.673248,0.30222,0.646493,-0.193511],[0,0,0,1],[9E+9,9E+9,9E+9,9E+9,9E+9,9E+9]];
CONST robtarget H_p4up:=[[-143.89,-150.66,48.7],[0.673248,0.30222,0.646493,-0.193511],[0,0,0,1],[9E+09,9E+09,9E+09,9E+09,9E+09,9E+09]];
CONST robtarget H_p4up10:=[[-110.25,-120.75,34.42],[0.673248,0.302219,0.646494,-0.193511],[0,0,0,1],[9E+9,9E+9,9E+9,9E+9,9E+9,9E+9]];
CONST robtarget H_p5:=[[-110.25,-120.75,34.42],[0.673248,0.302219,0.646494,-0.193511],[0,0,0,1],[9E+09,9E+09,9E+09,9E+09,9E+09,9E+09]];
CONST robtarget H_p15:=[[-117.03,-154.95,34.42],[0.673248,0.302219,0.646494,-0.193511],[0,0,0,1],[9E+9,9E+9,9E+9,9E+9,9E+9,9E+9]];
CONST robtarget H_p6:=[[-117.03,-154.95,34.42],[0.673248,0.302219,0.646494,-0.193511],[0,0,0,1],[9E+09,9E+09,9E+09,9E+09,9E+09,9E+09]];
CONST robtarget H_p16:=[[-117.03,-154.95,48.51],[0.673248,0.302219,0.646494,-0.193511],[0,0,0,1],[9E+9,9E+9,9E+9,9E+9,9E+9,9E+9]];
CONST robtarget H_p6up:=[[-117.03,-154.95,48.51],[0.673248,0.302219,0.646494,-0.193511],[0,0,0,1],[9E+09,9E+09,9E+09,9E+09,9E+09,9E+09]];
CONST robtarget H_p6up10:=[[-94.05,-174.96,61.34],[0.673248,0.302219,0.646494,-0.193511],[-1,0,0,1],[9E+9,9E+9,9E+9,9E+9,9E+9,9E+9]];
CONST robtarget R_p1up:=[[-94.05,-174.96,61.34],[0.673248,0.302219,0.646494,-0.193511],[-1,0,0,1],[9E+09,9E+09,9E+09,9E+09,9E+09,9E+09]];
CONST robtarget R_p1up10:=[[-94.05,-174.96,34.93],[0.673248,0.302219,0.646494,-0.193511],[-1,0,0,1],[9E+9,9E+9,9E+9,9E+9,9E+9,9E+9]];
CONST robtarget R_p1:=[[-94.05,-174.96,34.93],[0.673248,0.302219,0.646494,-0.193511],[-1,0,0,1],[9E+09,9E+09,9E+09,9E+09,9E+09,9E+09]];
CONST robtarget R_p11:=[[-146.07,-165.77,34.93],[0.673248,0.302219,0.646494,-0.193511],[-1,0,0,1],[9E+9,9E+9,9E+9,9E+9,9E+9,9E+9]];
CONST robtarget R_p2:=[[-146.07,-165.77,34.93],[0.673248,0.302219,0.646494,-0.193511],[-1,0,0,1],[9E+09,9E+09,9E+09,9E+09,9E+09,9E+09]];
CONST robtarget R_p12:=[[-145.81,-167.79,52.29],[0.673247,0.302219,0.646494,-0.193511],[-1,0,0,1],[9E+9,9E+9,9E+9,9E+9,9E+9,9E+9]];
CONST robtarget R_p2up:=[[-145.81,-167.79,52.29],[0.673247,0.302219,0.646494,-0.193511],[-1,0,0,1],[9E+09,9E+09,9E+09,9E+09,9E+09,9E+09]];
CONST robtarget R_p2up10:=[[-93.60,-174.98,34.89],[0.673247,0.302219,0.646495,-0.193511],[-1,0,0,1],[9E+9,9E+9,9E+9,9E+9,9E+9,9E+9]];
CONST robtarget R_p3:=[[-93.6,-174.98,34.89],[0.673247,0.302219,0.646495,-0.193511],[-1,0,0,1],[9E+09,9E+09,9E+09,9E+09,9E+09,9E+09]];
CONST robtarget R_p13:=[[-96.46,-191.20,34.89],[0.673247,0.30222,0.646495,-0.193511],[-1,0,0,1],[9E+9,9E+9,9E+9,9E+9,9E+9,9E+9]];
CONST robtarget R_p4:=[[-96.46,-191.2,34.89],[0.673247,0.30222,0.646495,-0.193511],[-1,0,0,1],[9E+09,9E+09,9E+09,9E+09,9E+09,9E+09]];
CONST robtarget R_p24:=[[-125.43,-184.72,34.89],[0.673247,0.30222,0.646495,-0.193511],[-1,0,0,1],[9E+9,9E+9,9E+9,9E+9,9E+9,9E+9]];
CONST robtarget R_p14:=[[-114.39,-200.92,34.89],[0.673247,0.30222,0.646495,-0.193511],[-1,0,0,1],[9E+9,9E+9,9E+9,9E+9,9E+9,9E+9]];
CONST robtarget R_p5:=[[-114.39,-200.92,34.89],[0.673247,0.30222,0.646495,-0.193511],[-1,0,0,1],[9E+09,9E+09,9E+09,9E+09,9E+09,9E+09]];
CONST robtarget R_p6:=[[-125.43,-184.72,34.89],[0.673247,0.30222,0.646495,-0.193511],[-1,0,0,1],[9E+09,9E+09,9E+09,9E+09,9E+09,9E+09]];
CONST robtarget R_p15:=[[-122.84,-170.06,34.89],[0.673247,0.30222,0.646494,-0.193511],[-1,0,0,1],[9E+9,9E+9,9E+9,9E+9,9E+9,9E+9]];
CONST robtarget R_p7:=[[-122.84,-170.06,34.89],[0.673247,0.30222,0.646494,-0.193511],[-1,0,0,1],[9E+09,9E+09,9E+09,9E+09,9E+09,9E+09]];
CONST robtarget R_p17:=[[-125.49,-185.05,35.71],[0.673247,0.30222,0.646495,-0.193511],[-1,0,0,1],[9E+9,9E+9,9E+9,9E+9,9E+9,9E+9]];
CONST robtarget R_p8:=[[-125.49,-185.05,35.71],[0.673247,0.30222,0.646495,-0.193511],[-1,0,0,1],[9E+09,9E+09,9E+09,9E+09,9E+09,9E+09]];
CONST robtarget R_p18:=[[-151.35,-194.66,35.72],[0.673248,0.30222,0.646494,-0.19351],[-1,0,0,1],[9E+9,9E+9,9E+9,9E+9,9E+9,9E+9]];
CONST robtarget R_p9:=[[-151.35,-194.66,35.72],[0.673248,0.30222,0.646494,-0.19351],[-1,0,0,1],[9E+09,9E+09,9E+09,9E+09,9E+09,9E+09]];
CONST robtarget R_p19:=[[-151.35,-194.66,58.90],[0.673248,0.30222,0.646494,-0.193511],[-1,0,0,1],[9E+9,9E+9,9E+9,9E+9,9E+9,9E+9]];
CONST robtarget R_endup:=[[-151.35,-194.66,58.9],[0.673248,0.30222,0.646494,-0.193511],[-1,0,0,1],[9E+09,9E+09,9E+09,9E+09,9E+09,9E+09]];
CONST robtarget R_endup10:=[[-101.79,-214.77,59.03],[0.673248,0.302219,0.646494,-0.193511],[-1,0,0,1],[9E+9,9E+9,9E+9,9E+9,9E+9,9E+9]];
CONST robtarget I_strtup:=[[-101.79,-214.77,59.03],[0.673248,0.302219,0.646494,-0.193511],[-1,0,0,1],[9E+09,9E+09,9E+09,9E+09,9E+09,9E+09]];
CONST robtarget I_strtup10:=[[-101.79,-214.77,34.79],[0.673248,0.302219,0.646494,-0.193511],[-1,0,0,1],[9E+9,9E+9,9E+9,9E+9,9E+9,9E+9]];
CONST robtarget I_p1:=[[-101.79,-214.77,34.79],[0.673248,0.302219,0.646494,-0.193511],[-1,0,0,1],[9E+09,9E+09,9E+09,9E+09,9E+09,9E+09]];
CONST robtarget I_p11:=[[-152.67,-205.50,34.79],[0.673248,0.302219,0.646494,-0.193511],[-1,0,0,1],[9E+9,9E+9,9E+9,9E+9,9E+9,9E+9]];
CONST robtarget I_p2:=[[-152.67,-205.5,34.79],[0.673248,0.302219,0.646494,-0.193511],[-1,0,0,1],[9E+09,9E+09,9E+09,9E+09,9E+09,9E+09]];
CONST robtarget I_p12:=[[-152.67,-205.50,56.28],[0.673248,0.302219,0.646494,-0.193511],[-1,0,0,1],[9E+9,9E+9,9E+9,9E+9,9E+9,9E+9]];
CONST robtarget I_p2up:=[[-152.67,-205.5,56.28],[0.673248,0.302219,0.646494,-0.193511],[-1,0,0,1],[9E+09,9E+09,9E+09,9E+09,9E+09,9E+09]];
CONST robtarget I_p2up10:=[[-118.47,-257.29,53.39],[0.673248,0.302219,0.646494,-0.193511],[-1,0,0,1],[9E+9,9E+9,9E+9,9E+9,9E+9,9E+9]];
CONST robtarget S_p1:=[[-118.47,-257.29,53.39],[0.673248,0.302219,0.646494,-0.193511],[-1,0,0,1],[9E+9,9E+9,9E+9,9E+9,9E+9,9E+9]];
CONST robtarget S_p1up:=[[-118.47,-257.29,53.61],[0.673248,0.302219,0.646494,-0.19351],[-1,0,0,1],[9E+09,9E+09,9E+09,9E+09,9E+09,9E+09]];
CONST robtarget S_p1up10:=[[-118.47,-257.29,34.48],[0.673248,0.302219,0.646494,-0.19351],[-1,0,0,1],[9E+9,9E+9,9E+9,9E+9,9E+9,9E+9]];
CONST robtarget S_p1strt:=[[-118.47,-257.29,34.48],[0.673248,0.302219,0.646494,-0.19351],[-1,0,0,1],[9E+09,9E+09,9E+09,9E+09,9E+09,9E+09]];
CONST robtarget S_p1strt20:=[[-106.06,-235.68,34.48],[0.673248,0.302219,0.646495,-0.19351],[-1,0,0,1],[9E+9,9E+9,9E+9,9E+9,9E+9,9E+9]];
CONST robtarget S_p1strt10:=[[-106.06,-235.68,34.48],[0.673248,0.302219,0.646495,-0.19351],[-1,0,0,1],[9E+9,9E+9,9E+9,9E+9,9E+9,9E+9]];
CONST robtarget S_p2:=[[-106.06,-235.68,34.48],[0.673248,0.302219,0.646495,-0.19351],[-1,0,0,1],[9E+09,9E+09,9E+09,9E+09,9E+09,9E+09]];
CONST robtarget S_p3:=[[-128.84,-233.05,34.48],[0.673248,0.302219,0.646494,-0.19351],[-1,0,0,1],[9E+09,9E+09,9E+09,9E+09,9E+09,9E+09]];
CONST robtarget S_p12:=[[-135.23,-244.09,34.48],[0.673248,0.302219,0.646494,-0.19351],[-1,0,0,1],[9E+9,9E+9,9E+9,9E+9,9E+9,9E+9]];
CONST robtarget S_p4:=[[-135.23,-244.09,34.48],[0.673248,0.302219,0.646494,-0.19351],[-1,0,0,1],[9E+09,9E+09,9E+09,9E+09,9E+09,9E+09]];
CONST robtarget S_p24:=[[-144.42,-219.97,34.48],[0.673249,0.302219,0.646494,-0.19351],[-1,0,0,1],[9E+9,9E+9,9E+9,9E+9,9E+9,9E+9]];
CONST robtarget S_p14:=[[-158.43,-242.54,34.48],[0.673248,0.302219,0.646494,-0.19351],[-1,0,0,1],[9E+9,9E+9,9E+9,9E+9,9E+9,9E+9]];
CONST robtarget S_p5:=[[-158.43,-242.54,34.48],[0.673248,0.302219,0.646494,-0.19351],[-1,0,0,1],[9E+09,9E+09,9E+09,9E+09,9E+09,9E+09]];
CONST robtarget S_p6:=[[-144.42,-219.97,34.48],[0.673249,0.302219,0.646494,-0.19351],[-1,0,0,1],[9E+09,9E+09,9E+09,9E+09,9E+09,9E+09]];
CONST robtarget S_p15:=[[-144.42,-219.97,51.82],[0.673249,0.302219,0.646493,-0.19351],[-1,0,0,1],[9E+9,9E+9,9E+9,9E+9,9E+9,9E+9]];
CONST robtarget S_p6up:=[[-144.42,-219.97,51.82],[0.673249,0.302219,0.646493,-0.19351],[-1,0,0,1],[9E+9,9E+9,9E+9,9E+9,9E+9,9E+9]];
CONST robtarget S_p6endindup:=[[-144.42,-219.97,51.82],[0.673249,0.302219,0.646493,-0.19351],[-1,0,0,1],[9E+09,9E+09,9E+09,9E+09,9E+09,9E+09]];
CONST robtarget S_p6endindup10:=[[-5.46,-204.24,119.19],[0.67325,0.302219,0.646492,-0.19351],[-1,0,0,1],[9E+9,9E+9,9E+9,9E+9,9E+9,9E+9]];
CONST robtarget endmove1:=[[-5.46,-204.24,119.19],[0.67325,0.302219,0.646492,-0.19351],[-1,0,0,1],[9E+09,9E+09,9E+09,9E+09,9E+09,9E+09]];
CONST robtarget endmove11:=[[-1.77,-151.13,108.48],[0.658161,0.135707,0.74048,-0.00981134],[-1,-1,0,1],[9E+9,9E+9,9E+9,9E+9,9E+9,9E+9]];
CONST robtarget endmove2:=[[-1.77,-151.13,108.48],[0.658161,0.135707,0.74048,-0.00981134],[-1,-1,0,1],[9E+09,9E+09,9E+09,9E+09,9E+09,9E+09]];
CONST robtarget endmove12:=[[61.72,-121.56,235.27],[0.745809,0.0892119,0.65999,0.0149501],[0,-1,0,1],[9E+9,9E+9,9E+9,9E+9,9E+9,9E+9]];
CONST robtarget lastmove:=[[61.72,-121.56,235.27],[0.745809,0.0892119,0.65999,0.0149501],[0,-1,0,1],[9E+09,9E+09,9E+09,9E+09,9E+09,9E+09]];
VAR num MyChoice_:=0;
    !***********************************************************
    !
    ! Module:  Module1
    !
    ! Description:
    !   <Insert description here>
    !
    ! Author: hp
    !
    ! Version: 1.0
    !
    !***********************************************************


    !***********************************************************
    !
    ! Procedure main
    !
    !   This is the entry point of your program
    !
    !***********************************************************
    PROC main()
        TPErase;
        TPWrite "Drawing Demo";
        TPReadFK MyChoice, "What do you want to write or draw?", "Square", "D_Shape", "Circle", "Salford", "MyName";
        TEST MyChoice
        CASE 1:
         Square;
        CASE 2:
         D_Shape;
        CASE 3:
         Circle;
        CASE 4:
         Salford;
        CASE 5:
         MyName;
        ENDTEST
    ENDPROC
PROC Square()
        MoveJ startpoint, v100, z50, toolpen\WObj:=wobjshapes;
        MoveJ stp_sqr, v100, z50, toolpen\WObj:=wobjshapes;
        MoveL sqr1, v100, fine, toolpen\WObj:=wobjshapes;
        MoveL sqr2, v100, fine, toolpen\WObj:=wobjshapes;
        MoveL sqr3, v100, fine, toolpen\WObj:=wobjshapes;
        MoveL sqr4, v100, fine, toolpen\WObj:=wobjshapes;
        MoveL sqr5, v100, fine, toolpen\WObj:=wobjshapes;
        MoveL sqr_end_up, v100, z50, toolpen\WObj:=wobjshapes;
ENDPROC
PROC D_Shape()
        WaitTime 2;
        MoveJ Dshp_start_up, v100, z50, toolpen\WObj:=wobjshapes;
        MoveL Dshp_pt1, v100, z50, toolpen\WObj:=wobjshapes;
        MoveL Dshp_pt2, v100, z50, toolpen\WObj:=wobjshapes;
        MoveL Dshp_pt3, v100, z50, toolpen\WObj:=wobjshapes;
        MoveC Dshp_crv1, Dshp_crv2, v100, z10, toolpen\WObj:=wobjshapes;
        MoveL Dshp_pt4, v100, fine, toolpen\WObj:=wobjshapes;
        MoveL Dshp_end_up, v100, z50, toolpen\WObj:=wobjshapes;
ENDPROC
PROC Circle()
        WaitTime 2;
        MoveL Crcl_start_up, v100, z50, toolpen\WObj:=wobjshapes;
        MoveL Crcl_start_pt1, v100, z50, toolpen\WObj:=wobjshapes;
        MoveC Crcl_pt2, Crcl_pt3, v100, z10, toolpen\WObj:=wobjshapes;
        MoveC Crcl_pt4, Crcl_pt5, v100, z10, toolpen\WObj:=wobjshapes;
        MoveL Crcl_end_up, v100, z50, toolpen\WObj:=wobjshapes;
        WaitTime 2;
ENDPROC
PROC Salford()
        MoveL S_pt1_up, v100, z50, toolpen\WObj:=wobjsalf;
        MoveL S_pt1_dwn, v100, fine, toolpen\WObj:=wobjsalf;
        MoveC S_pt2_crv, S_pt3_crv2, v100, fine, toolpen\WObj:=wobjsalf;
        MoveL S_pt4, v100, z50, toolpen\WObj:=wobjsalf;
        MoveC S_pt5_crv3, S_pt6_crv4, v100, fine, toolpen\WObj:=wobjsalf;
        MoveL S_end_up, v100, fine, toolpen\WObj:=wobjsalf;
        MoveL A_start_up, v100, z50, toolpen\WObj:=wobjsalf;
        MoveL A_start_pt1, v100, fine, toolpen\WObj:=wobjsalf;
        MoveL A_pt2, v100, fine, toolpen\WObj:=wobjsalf;
        MoveL A_line1_up, v100, fine, toolpen\WObj:=wobjsalf;
        MoveL A_line2_strt, v100, fine, toolpen\WObj:=wobjsalf;
        MoveL A_line2_stp, v100, fine, toolpen\WObj:=wobjsalf;
        MoveL A_line2_endup, v100, fine, toolpen\WObj:=wobjsalf;
        MoveL A_crssline_up, v100, fine, toolpen\WObj:=wobjsalf;
        MoveL A_crssline_pt1, v100, fine, toolpen\WObj:=wobjsalf;
        MoveL A_crssline_pt2, v100, fine, toolpen\WObj:=wobjsalf;
        MoveL A_end_up, v100, z50, toolpen\WObj:=wobjsalf;
        MoveL L_start_up, v100, fine, toolpen\WObj:=wobjsalf;
        MoveL L_start_pt1, v100, fine, toolpen\WObj:=wobjsalf;
        MoveL L_pt3_dwn, v100, fine, toolpen\WObj:=wobjsalf;
        MoveL L_end_pt4, v100, fine, toolpen\WObj:=wobjsalf;
        MoveL L_end_ptup, v100, fine, toolpen\WObj:=wobjsalfs;
        MoveL F_pt1_up, v100, z50, toolpen\WObj:=wobjsalf;
        MoveL F_pt1_dwn, v100, fine, toolpen\WObj:=wobjsalf;
        MoveL F_pt2, v100, fine, toolpen\WObj:=wobjsalf;
        MoveL F_pt3, v100, fine, toolpen\WObj:=wobjsalf;
        MoveL F_pt4, v100, fine, toolpen\WObj:=wobjsalfs;
        MoveL F_pt5, v100, fine, toolpen\WObj:=wobjsalf;
        MoveL F_pt5_up, v100, fine, toolpen\WObj:=wobjsalf;
        MoveL F_pt6, v100, fine, toolpen\WObj:=wobjsalf;
        MoveL F_pt7_enddwn, v100, fine, toolpen\WObj:=wobjsalf;
        MoveL F_pt7_endup, v100, z50, toolpen\WObj:=wobjsalf;
        MoveL O_pt1_strtup, v100, z50, toolpen\WObj:=wobjsalf;
        MoveL O_pt1_dwn, v100, fine, toolpen\WObj:=wobjsalf;
        MoveC O_crv1, O_crv2, v100, fine, toolpen\WObj:=wobjsalf;
        MoveL O_pt2, v100, fine, toolpen\WObj:=wobjsalf;
        MoveC O_crv3, O_crv4, v100, fine, toolpen\WObj:=wobjsalf;
        MoveL O_endpt_dwn, v100, fine, toolpen\WObj:=wobjsalf;
        MoveL O_endpt_up, v100, z50, toolpen\WObj:=wobjsalf;
        MoveL R_strtpt_up, v100, z50, toolpen\WObj:=wobjsalf;
        MoveL R_strt_pt1, v100, fine, toolpen\WObj:=wobjsalf;
        MoveL R_pt2, v100, fine, toolpen\WObj:=wobjsalf;
        MoveL R_crvpt1, v100, fine, toolpen\WObj:=wobjsalf;
        MoveC R_crvpt2, R_crvpt3, v100, fine, toolpen\WObj:=wobjsalf;
        MoveL R_endline1, v100, fine, toolpen\WObj:=wobjsalf;
        MoveL R_endline2, v100, fine, toolpen\WObj:=wobjsalf;
        MoveL R_endline_up, v100, z50, toolpen\WObj:=wobjsalf;
        MoveL D_strt_up, v100, z50, toolpen\WObj:=wobjsalf;
        MoveL D_pt1, v100, fine, toolpen\WObj:=wobjsalf;
        MoveL D_pt2, v100, fine, toolpen\WObj:=wobjsalf;
        MoveC D_crvpt1, D_crvpt2_end, v100, fine, toolpen\WObj:=wobjsalf;
        MoveL D_end_up, v100, z50, toolpen\WObj:=wobjsalf;
        WaitTime 2;
ENDPROC
PROC MyName()
        MoveL Name_strtpt_up, v100, z50, toolpen\WObj:=wobjname;
        MoveL C_pt1, v100, z50, toolpen\WObj:=wobjname;
        MoveC C_pt2, C_pt3, v100, fine, toolpen\WObj:=wobjname;
        MoveL C_p4, v100, fine, toolpen\WObj:=wobjname;
        MoveC C_p5, C_p6, v100, fine, toolpen\WObj:=wobjname;
        MoveL C_end_up, v100, fine, toolpen\WObj:=wobjname;
        MoveL H_startup, v100, fine, toolpen\WObj:=wobjname;
        MoveL H_pt1, v100, fine, toolpen\WObj:=wobjnames;
        MoveL H_pt2, v100, fine, toolpen\WObj:=wobjname;
        MoveL H_p2up, v100, fine, toolpen\WObj:=wobjname;
        MoveL H_p3up, v100, fine, toolpen\WObj:=wobjname;
        MoveL H_p3, v100, fine, toolpen\WObj:=wobjname;
        MoveL H_p4, v100, fine, toolpen\WObj:=wobjname;
        MoveL H_p4up, v100, fine, toolpen\WObj:=wobjname;
        MoveL H_p5, v100, fine, toolpen\WObj:=wobjnames;
        MoveL H_p6, v100, fine, toolpen\WObj:=wobjname;
        MoveL H_p6up, v100, fine, toolpen\WObj:=wobjname;
        MoveL R_p1up, v100, fine, toolpen\WObj:=wobjnames;
        MoveL R_p1, v100, fine, toolpen\WObj:=wobjname;
        MoveL R_p2, v100, fine, toolpen\WObj:=wobjname;
        MoveL R_p2up, v100, fine, toolpen\WObj:=wobjnames;
        MoveL R_p3, v100, fine, toolpen\WObj:=wobjname;
        MoveL R_p4, v100, fine, toolpen\WObj:=wobjname;
        MoveC R_p5, R_p6, v100, fine, toolpen\WObj:=wobjname;
        MoveL R_p7, v100, fine, toolpen\WObj:=wobjname;
        MoveL R_p8, v100, fine, toolpen\WObj:=wobjname;
        MoveL R_p9, v100, fine, toolpen\WObj:=wobjname;
        MoveL R_endup, v100, fine, toolpen\WObj:=wobjname;
        MoveL I_strtup, v100, fine, toolpen\WObj:=wobjname;
        MoveL I_p1, v100, fine, toolpen\WObj:=wobjname;
        MoveL I_p2, v100, fine, toolpen\WObj:=wobjname;
        MoveL I_p2up, v100, fine, toolpen\WObj:=wobjname;
        MoveL S_p1up, v100, fine, toolpen\WObj:=wobjname;
        MoveL S_p1strt, v100, fine, toolpen\WObj:=wobjname;
        MoveC S_p2, S_p3, v100, fine, toolpen\WObj:=wobjname;
        MoveL S_p4, v100, fine, toolpen\WObj:=wobjname;
        MoveC S_p5, S_p6, v100, fine, toolpen\WObj:=wobjname;
        MoveL S_p6endindup, v100, fine, toolpen\WObj:=wobjname;
        WaitTime 2;
        MoveL endmove1, v100, fine, toolpen\WObj:=wobjname;
        MoveL endmove2, v100, fine, toolpen\WObj:=wobjname;
        MoveL lastmove, v100, fine, toolpen\WObj:=wobjname;
ENDPROC
ENDMODULE
